INTERFACE ITcaCarrier

METHOD ChangeData : ITcoTaskStatus 
VAR_INPUT
	inData : TcaCarrierData;
END_VAR
END_METHOD

METHOD CoordinatesOf : ST_Coordinate
VAR_INPUT
	WorkpiecePlace		: INT;
END_VAR
END_METHOD

METHOD CountEmptyPlaces : INT
END_METHOD

METHOD CountPlacesByStatus : INT
VAR_INPUT
	nStatus			: INT;
END_VAR
END_METHOD

METHOD FillWithWorkpieces_CustomStatus : ITcoTaskStatus
VAR_INPUT
	Status		: eTcaWorkpiecePlaceStatus;
END_VAR
END_METHOD

METHOD FillWithWorkpieces_InitialStatus : ITcoTaskStatus
VAR_INPUT
END_VAR
END_METHOD

METHOD FillWithWorkpieces_RequestStatus : ITcoTaskStatus
VAR_INPUT
END_VAR
END_METHOD

METHOD FindPlace : REFERENCE TO TcaWorkpiecePlace //-1..no Position found

VAR_INPUT
	Status		: eTcaWorkpiecePlaceStatus;
END_VAR
END_METHOD

METHOD GetPlaceReference : REFERENCE TO TcaWorkpiecePlace
VAR_INPUT
	nIndexNr		: INT;
END_VAR
END_METHOD

METHOD RefreshStatus : BOOL
END_METHOD

END_INTERFACE

(* stored: Version 1.1.0.1
   Itf ITcaCarrier: Id {9e0cc9a0-5bab-475e-9e88-b5fff12293c9}
   Folder Functions: Id {1e800a71-c285-4ec9-9aa6-ecbd6bf9086d}
   Folder Operations: Id {30674b05-788f-4a94-9200-886c1882f18d}
   Method ChangeData: Id {2a55adf0-b717-49e0-a848-988923e4f914}
   Method CoordinatesOf: Id {353b1b64-e9b2-4b07-b088-df984ca08abb}
   Method CountEmptyPlaces: Id {435ff8d8-5c92-4d60-8b6a-16590e4a2b4f}
   Method CountPlacesByStatus: Id {dc1e3558-9357-40d6-ae2b-69783cdf18c8}
   Method FillWithWorkpieces_CustomStatus: Id {4acdadd2-be97-494c-acce-ffdb37c9c70a}
   Method FillWithWorkpieces_InitialStatus: Id {605f3eb6-38ee-413e-aa90-8877d2b07d06}
   Method FillWithWorkpieces_RequestStatus: Id {581aa0bb-30b5-4f4b-98b6-6be31673be6c}
   Method FindPlace: Id {9e1f683f-bc34-41fe-9ad4-ad4cf83ca3f4}
   Method GetPlaceReference: Id {b4a1ebfa-681f-488c-a804-1d0346bbae1f}
   Method RefreshStatus: Id {5eb8017c-eecb-44c7-a338-9771d947a54d} *)
